TYPE E_DriverCtrlWord :
(
	DriverCtrlWord_INIT := 6,
	DriverCtrlWord_PREOP := 7,
	DriverCtrlWord_OP := 15,
	DriverCtrlWord_FaultReset := 16#80,
	DriverCtrlWord_halt := 16#10F
);
END_TYPE

(* stored: Version 1.1.0.1, ProductVersion 3.1.4024.12
   DUT E_DriverCtrlWord: Id {d6673421-3c73-4541-ae90-0a167e8564dd} *)
